    {attribute 'pytmc' := 'pv: TOP:RTD:01'}
    RTD_TOP_1 : FB_CC_TempSensor;
    {attribute 'pytmc' := 'pv: TOP:RTD:02'}
    RTD_TOP_2 : FB_CC_TempSensor;
    {attribute 'pytmc' := 'pv: BOTTOM:RTD:01'}
    RTD_Bottom_1 : FB_CC_TempSensor;
    {attribute 'pytmc' := 'pv: BOTTOM:RTD:02'}
    RTD_Bottom_2 : FB_CC_TempSensor;
    {attribute 'pytmc' := 'pv: NORTH:RTD:01'}
    RTD_North_1 : FB_CC_TempSensor;
    {attribute 'pytmc' := 'pv: NORTH:RTD:02'}
    RTD_North_2 : FB_CC_TempSensor;
    {attribute 'pytmc' := 'pv: SOUTH:RTD:01'}
    RTD_South_1 : FB_CC_TempSensor;
    {attribute 'pytmc' := 'pv: SOUTH:RTD:02'}
    RTD_South_2 : FB_CC_TempSensor;
    (* PMPS reactive-DB key for the device's allowed temperature. *)
    sPmpsState : STRING;
    fbReadPMPSDB : FB_JsonDocToSafeBP;
    astTempDB    : ARRAY[1..1] OF ST_DbStateParams;
    (* fbReadPMPSDB.bExecute needs a rising edge; a real PMPS file read produces one as bBusy falls.
       Taken as REFERENCE TO so a test can drive its own BOOL and simulate the edge
       instead of reaching into MOTION_GVL.fbPmpsFileReader directly.
    *)
    bFileReaderBusy : REFERENCE TO BOOL;
    (* Margin (mm) subtracted from the authorized width/height when snapping
       the request into PMPS compliance. Set via FB_Init, defaults to 0.01. *)
    fApertureMargin : REAL := 0.01;
END_VAR

IF NOT __ISVALIDREF(THIS^.aiMotionStage)
   OR NOT __ISVALIDREF(THIS^.fbFFHWO) OR NOT __ISVALIDREF(bFileReaderBusy) THEN
    RETURN;
END_IF


// Parent body: EPICS edge-trigger consumption only (no REF touch).
SUPER^();


// Inherited dispatch (parity with legacy FB_SLITS_POWER body
// invoking ACT_CalculatePositions / ACT_Motion).
M_CalculatePositions();
M_Motion();

// PMPS reactive temperature DB lookup. bExecute needs a rising edge,
// produced as the caller-injected file-reader busy flag falls. Guard
// the REF (single condition, no short-circuit hazard) so an unbound
// instance stays inert rather than dereferencing a nil ref.
astTempDB[1].sPmpsState := sPmpsState;
fbReadPMPSDB(
    bExecute    := NOT bFileReaderBusy,
    jsonDoc     := PMPS_GVL.BP_jsonDoc,
    sDeviceName := sDeviceName,
    arrStates   := astTempDB,
    io_fbFFHWO  := fbFFHWO
);

// All 8 RTDs share the same fault threshold (resolved from the DB).
RTD_TOP_1(
    fFaultThreshold := astTempDB[1].stReactiveParams.nTempSP,
    sDevName        := sDeviceName,
    io_fbFFHWO      := fbFFHWO
);
RTD_TOP_2(
    fFaultThreshold := astTempDB[1].stReactiveParams.nTempSP,
    sDevName        := sDeviceName,
    io_fbFFHWO      := fbFFHWO
);
RTD_Bottom_1(
    fFaultThreshold := astTempDB[1].stReactiveParams.nTempSP,
    sDevName        := sDeviceName,
    io_fbFFHWO      := fbFFHWO
);
RTD_Bottom_2(
    fFaultThreshold := astTempDB[1].stReactiveParams.nTempSP,
    sDevName        := sDeviceName,
    io_fbFFHWO      := fbFFHWO
);
RTD_North_1(
    fFaultThreshold := astTempDB[1].stReactiveParams.nTempSP,
    sDevName        := sDeviceName,
    io_fbFFHWO      := fbFFHWO
);
RTD_North_2(
    fFaultThreshold := astTempDB[1].stReactiveParams.nTempSP,
    sDevName        := sDeviceName,
    io_fbFFHWO      := fbFFHWO
);
RTD_South_1(
    fFaultThreshold := astTempDB[1].stReactiveParams.nTempSP,
    sDevName        := sDeviceName,
    io_fbFFHWO      := fbFFHWO
);
RTD_South_2(
    fFaultThreshold := astTempDB[1].stReactiveParams.nTempSP,
    sDevName        := sDeviceName,
    io_fbFFHWO      := fbFFHWO
);

fbFlowSwitch();

(* Records sPmpsState and REF-binds the caller-owned file-reader busy flag;
   aiMotionStage (4 blades), fbFFHWO and sDeviceName are bound by base
   FB_SLITS.FB_Init. Blade wiring runs from CallAfterInit. *)
{attribute 'analysis' := '-33'}
METHOD FB_Init : BOOL
VAR_INPUT
    bInitRetains  : BOOL;
    bInCopyCode   : BOOL;
    aiMotionStage : REFERENCE TO ARRAY[1..4] OF I_MotionStage;
    fbFFHWO       : REFERENCE TO FB_HardwareFFOutput;
    sDeviceName   : STRING;
    sPmpsState 	  : STRING;
    bFileReaderBusy : REFERENCE TO BOOL;
    fApertureMargin : REAL;
END_VAR
THIS^.sPmpsState := sPmpsState;
THIS^.bFileReaderBusy REF= bFileReaderBusy;
THIS^.fApertureMargin := fApertureMargin;
END_METHOD

(* Integrator-driven PMPS aperture-safety reconciliation, called each cycle
   with index = this device's slot in astApertures. Mirrors actual geometry
   into AptArrayStatus, faults FFO when actual gap exceeds the authorized
   envelope (or always, out of PMPS mode), and in PMPS mode snaps the request
   into compliance. Caller must ensure index is valid (no short-circuit). *)
METHOD M_UpdatePMPS : BOOL
VAR_INPUT
    index : INT;
END_VAR
// Mirror current actual aperture geometry and any-blade error state.
THIS^.AptArrayStatus.Height := THIS^.rActApertureSizeY;
THIS^.AptArrayStatus.Width  := THIS^.rActApertureSizeX;
THIS^.AptArrayStatus.xOK    :=
        NOT (THIS^.aiMotionStage[E_SlitsBlade.TOP   ].MotionStatus.bError)
    AND NOT (THIS^.aiMotionStage[E_SlitsBlade.BOTTOM].MotionStatus.bError)
    AND NOT (THIS^.aiMotionStage[E_SlitsBlade.NORTH ].MotionStatus.bError)
    AND NOT (THIS^.aiMotionStage[E_SlitsBlade.SOUTH ].MotionStatus.bError);

// Aperture-envelope evaluation.
IF ( THIS^.rActApertureSizeX > (AptArrayReq.Width  - (2 * ABS(THIS^.rActCenterX)))
     AND PMPS_GVL.stCurrentBeamParameters.astApertures[index].Width  > 0 )
OR ( THIS^.rActApertureSizeY > (AptArrayReq.Height - (2 * ABS(THIS^.rActCenterY)))
     AND PMPS_GVL.stCurrentBeamParameters.astApertures[index].Height > 0 ) THEN
    FFO.i_xOK := FALSE;
ELSE
    FFO.i_xOK := TRUE;
END_IF

IF xPMPSMode THEN
    IF THIS^.rActApertureSizeX > AptArrayReq.Width THEN
        rReqApertureSizeX := AptArrayReq.Width - fApertureMargin;
    END_IF
    IF THIS^.rActApertureSizeY > AptArrayReq.Height THEN
        rReqApertureSizeY := AptArrayReq.Height - fApertureMargin;
    END_IF
ELSE
    FFO.i_xOK := FALSE;
END_IF

FFO(
    i_xAutoReset := TRUE,
    io_fbFFHWO   := fbFFHWO
);
END_METHOD

END_FUNCTION_BLOCK

// ---- Devices/SLITS/FB_SLITS.TcPOU
(* Four-blade slit aperture controller (Top/Bottom/North/South), ND framework.
   Each blade uses a per-cycle FB_StatePTPMove single-shot mover (targets
   recomputed from EPICS aperture width/center + encoder offsets), not a named
   state mover. Caller-owned stages, PMPS FFO and device name injected via FB_Init
   REFERENCE TO; CallAfterInit wires blade interfaces. Motion parameters
   (velocity/accel/decel/jerk) belong to the caller-owned stage, set once at
   commissioning and persisted; FB_SLITS does not apply them. *)
{attribute 'analysis' := '-33'}
{attribute 'call_after_init'}
FUNCTION_BLOCK FB_SLITS
VAR_INPUT
    {attribute 'pytmc' := '
    pv: PMPS_OK
    io: i
    field: ZNAM False
    field: ONAM True
    '}
    bMoveOk : BOOL;

    (* Per-blade encoder zero-offsets (EPICS-settable). *)
    {attribute 'pytmc' := '
    pv: Offset_Top
    io: io
    '}
    rEncoderOffsetTop : REAL;

    {attribute 'pytmc' := '
    pv: ZeroOffset_Bottom
    io: io
    '}
    rEncoderOffsetBottom : REAL;

    {attribute 'pytmc' := '
    pv: ZeroOffset_North
    io: io
    '}
    rEncoderOffsetNorth : REAL;

    {attribute 'pytmc' := '
    pv: ZeroOffset_South
    io: io
    '}
    rEncoderOffsetSouth : REAL;
END_VAR
VAR CONSTANT
    (* Position-compare deltas for the blade ST_PositionState. *)
    fSmallDelta : LREAL := 0.01;
     (* Reference blade motion tuning (velocity/accel/decel/jerk). Not applied
       here: motion parameters belong to the caller-owned stage, set once at
       commissioning and persisted. Kept as commissioning reference values. *)
    // fVelocity     : LREAL := 0.2;
    // fAcceleration : LREAL := 0.8;
    // fDeceleration : LREAL := 0.8;
    // fJerk         : LREAL := 0.0;
END_VAR
VAR
    (* Per-blade scratch ST_PositionState. Static fields seeded here;
       fPosition and bMoveOk are refreshed each cycle in the body. *)
    stTop    : ST_PositionState := (sName := 'Top',    bValid := TRUE, bUseRawCounts := FALSE, fDelta := fSmallDelta);
    stBottom : ST_PositionState := (sName := 'Bottom', bValid := TRUE, bUseRawCounts := FALSE, fDelta := fSmallDelta);
    stNorth  : ST_PositionState := (sName := 'North',  bValid := TRUE, bUseRawCounts := FALSE, fDelta := fSmallDelta);
    stSouth  : ST_PositionState := (sName := 'South',  bValid := TRUE, bUseRawCounts := FALSE, fDelta := fSmallDelta);

    (* Per-blade PTP movers. iMotionStage is wired in CallAfterInit;
       FB_StatePTPMove tolerates a nil interface until then. *)
    {attribute 'pytmc' := 'pv: TOP'}
    fbTop    : FB_StatePTPMove(
        stPositionState := stTop,
        iMotionStage:=0
    );
    {attribute 'pytmc' := 'pv: BOTTOM'}
    fbBottom : FB_StatePTPMove(
        stPositionState := stBottom,
        iMotionStage:=0
    );
    {attribute 'pytmc' := 'pv: NORTH'}
    fbNorth  : FB_StatePTPMove(
        stPositionState := stNorth,
        iMotionStage:=0
    );
    {attribute 'pytmc' := 'pv: SOUTH'}
    fbSouth  : FB_StatePTPMove(
        stPositionState := stSouth,
        iMotionStage:=0
    );

    (* Aperture-math intermediate targets. *)
    fPosTopBlade    : LREAL;
    fPosBottomBlade : LREAL;
    fPosNorthBlade  : LREAL;
    fPosSouthBlade  : LREAL;

    (* EPICS request / actual aperture geometry. *)
    {attribute 'pytmc' := '
    pv: XWID_REQ
    io: io
    '}
    rReqApertureSizeX : REAL;
    {attribute 'pytmc' := '
    pv: YWID_REQ
    io: io
    '}
    rReqApertureSizeY : REAL;
    {attribute 'pytmc' := '
    pv: XCEN_REQ
    io: io
    '}
    rReqCenterX : REAL;
    {attribute 'pytmc' := '
    pv: YCEN_REQ
    io: io
    '}
    rReqCenterY : REAL;

    {attribute 'pytmc' := '
    pv: ACTUAL_XWIDTH
    io: io
    '}
    rActApertureSizeX : REAL;
    {attribute 'pytmc' := '
    pv: ACTUAL_YWIDTH
    io: io
    '}
    rActApertureSizeY : REAL;
    {attribute 'pytmc' := '
    pv: ACTUAL_XCENTER
    io: io
    '}
    rActCenterX : REAL;
    {attribute 'pytmc' := '
    pv: ACTUAL_YCENTER
    io: io
    '}
    rActCenterY : REAL;

    (* Edge-trigger request flags. Cleared on the rising edge each
       cycle but no preset move is dispatched (stub: legacy parity). *)
    {attribute 'pytmc' := '
    pv: OPEN
    io: io
    field: ZNAM False
    field: ONAM True
    '}
    bOpen : BOOL;

    {attribute 'pytmc' := '
    pv: CLOSE
    io: io
    field: ZNAM False
    field: ONAM True
    '}
    bClose : BOOL;

    {attribute 'pytmc' := '
    pv: BLOCK
    io: io
    field: ZNAM False
    field: ONAM True
    '}
    bBlock : BOOL;

    rTrig_Block : R_TRIG;
    rTrig_Open  : R_TRIG;
    rTrig_Close : R_TRIG;

    (* Change-detection latches for EPICS request fields. *)
    rOldReqApertureSizeX : REAL;
    rOldReqApertureSizeY : REAL;
    rOldReqCenterX       : REAL;
    rOldReqCenterY       : REAL;

    bExecuteMotionX : BOOL;
    bExecuteMotionY : BOOL;

    fbLogger : FB_LogMessage := (eSubsystem := E_SubSystem.MOTION);

    (* PMPS aperture-safety fault (driven by FB_SLITS_POWER.M_UpdatePMPS). *)
    FFO : FB_FastFault := (
        i_DevName  := sDeviceName,
        i_Desc     := 'Fault occurs when gaps and/or centers are not within safe margins, or PMPS mode is switched OFF',
        i_TypeCode := 16#FAA
    );

    (* PMPS aperture IO (caller-mapped to terminals). *)
    AptArrayStatus AT %Q* : ST_PMPS_Aperture_IO;
    AptArrayReq    AT %I* : ST_PMPS_Aperture_IO;

    (* REF backing fields, populated by FB_Init. *)
    {attribute 'no_copy'}
    aiMotionStage : REFERENCE TO ARRAY[1..4] OF I_MotionStage;
    {attribute 'no_copy'}
    fbFFHWO       : REFERENCE TO FB_HardwareFFOutput;
    sDeviceName   :  STRING;
    nMotor : UINT;
END_VAR

// Legacy parity: the base body consumes only the EPICS Open / Close /
// Block edge-triggers. Blade init + motion dispatch lives on the
// FB_SLITS_POWER subclass body.
HandleRequests();

(* Auto-fired once after FB_Init binds the REFs. The four FB_StatePTPMove
   blade movers were inline-init'd with nil interface refs, so this re-supplies
   each blade's now-valid interface and scratch ST_PositionState, and sets the
   FFO device name. *)
{attribute 'call_after_init'}
METHOD CallAfterInit
fbTop.CallAfterInit(    stPositionState := stTop,    iMotionStage := aiMotionStage[E_SlitsBlade.TOP]);
fbBottom.CallAfterInit( stPositionState := stBottom, iMotionStage := aiMotionStage[E_SlitsBlade.BOTTOM]);
fbNorth.CallAfterInit(  stPositionState := stNorth,  iMotionStage := aiMotionStage[E_SlitsBlade.NORTH]);
fbSouth.CallAfterInit(  stPositionState := stSouth,  iMotionStage := aiMotionStage[E_SlitsBlade.SOUTH]);

FFO.i_DevName := sDeviceName;
END_METHOD

(* REF-binds caller-owned aiMotionStage (4 blades), fbFFHWO and sDeviceName
   at instantiation. Blade interface wiring runs from CallAfterInit once these
   REFs are bound. *)
{attribute 'analysis' := '-33'}
METHOD FB_Init : BOOL
VAR_INPUT
    bInitRetains  : BOOL;
    bInCopyCode   : BOOL;
    aiMotionStage : REFERENCE TO ARRAY[1..4] OF I_MotionStage;
    fbFFHWO       : REFERENCE TO FB_HardwareFFOutput;
    sDeviceName   : STRING;
END_VAR
THIS^.aiMotionStage REF= aiMotionStage;
THIS^.fbFFHWO       REF= fbFFHWO;
THIS^.sDeviceName   := sDeviceName;
END_METHOD

(*
    Consume the EPICS Open / Close / Block rising-edge requests and
    self-clear the flags. No preset move is dispatched (legacy stub).
*)
METHOD HandleRequests
rTrig_Block(CLK := bBlock);
rTrig_Open(CLK := bOpen);
rTrig_Close(CLK := bClose);

IF rTrig_Block.Q THEN
    bBlock := FALSE;
END_IF
IF rTrig_Open.Q THEN
    bOpen := FALSE;
END_IF
IF rTrig_Close.Q THEN
    bClose := FALSE;
END_IF
END_METHOD

(* Legacy ACT_CalculatePositions equivalent. Detects EPICS request changes
   (rejecting aperture sizes beyond the PMPS-authorized envelope), recomputes
   per-blade targets from requested gap + center + encoder offset, and refreshes
   actual aperture geometry feedback from caller-owned motor positions. *)
METHOD M_CalculatePositions
IF rOldReqApertureSizeX <> rReqApertureSizeX THEN
    IF rReqApertureSizeX <= AptArrayReq.Width THEN
        rOldReqApertureSizeX := rReqApertureSizeX;
        bExecuteMotionX      := TRUE;
        fbLogger(sMsg := 'Requested new X gap.', eSevr := TcEventSeverity.Verbose);
    ELSE
        fbLogger(
            sMsg := 'Requested new X gap is larger than PMPS request.',
            eSevr := TcEventSeverity.Verbose
        );
    END_IF
END_IF

IF rOldReqCenterX <> rReqCenterX THEN
    rOldReqCenterX  := rReqCenterX;
    bExecuteMotionX := TRUE;
    fbLogger(sMsg := 'Requested new X center', eSevr := TcEventSeverity.Verbose);
END_IF

IF rOldReqApertureSizeY <> rReqApertureSizeY THEN
    IF rReqApertureSizeY <= AptArrayReq.Height THEN
        rOldReqApertureSizeY := rReqApertureSizeY;
        bExecuteMotionY      := TRUE;
        fbLogger(sMsg := 'Requested new Y gap.', eSevr := TcEventSeverity.Verbose);
    ELSE
        fbLogger(
            sMsg := 'Requested new Y gap is larger than PMPS request.',
            eSevr := TcEventSeverity.Verbose
        );
    END_IF
END_IF

IF rOldReqCenterY <> rReqCenterY THEN
    rOldReqCenterY  := rReqCenterY;
    bExecuteMotionY := TRUE;
    fbLogger(sMsg := 'Requested new Y center.', eSevr := TcEventSeverity.Verbose);
END_IF

// Per-blade target positions from requested gap + center + per-blade
// encoder offset.
fPosTopBlade    :=  (rReqApertureSizeY / 2) + (rReqCenterY + rEncoderOffsetTop);
fPosBottomBlade := -(rReqApertureSizeY / 2) + (rReqCenterY + rEncoderOffsetBottom);
fPosNorthBlade  :=  (rReqApertureSizeX / 2) + (rReqCenterX + rEncoderOffsetNorth);
fPosSouthBlade  := -(rReqApertureSizeX / 2) + (rReqCenterX + rEncoderOffsetSouth);

// Actual aperture geometry feedback from caller-owned motors.
rActApertureSizeX := LREAL_TO_REAL(
    (aiMotionStage[E_SlitsBlade.NORTH].MotionStatus.fActPosition - rEncoderOffsetNorth)
  - (aiMotionStage[E_SlitsBlade.SOUTH].MotionStatus.fActPosition - rEncoderOffsetSouth)
);
rActApertureSizeY := LREAL_TO_REAL(
    (aiMotionStage[E_SlitsBlade.TOP].MotionStatus.fActPosition    - rEncoderOffsetTop)
  - (aiMotionStage[E_SlitsBlade.BOTTOM].MotionStatus.fActPosition - rEncoderOffsetBottom)
);
rActCenterX := LREAL_TO_REAL(
    ((aiMotionStage[E_SlitsBlade.NORTH].MotionStatus.fActPosition - rEncoderOffsetNorth)
   + (aiMotionStage[E_SlitsBlade.SOUTH].MotionStatus.fActPosition - rEncoderOffsetSouth)) / 2
);
rActCenterY := LREAL_TO_REAL(
    ((aiMotionStage[E_SlitsBlade.TOP].MotionStatus.fActPosition    - rEncoderOffsetTop)
   + (aiMotionStage[E_SlitsBlade.BOTTOM].MotionStatus.fActPosition - rEncoderOffsetBottom)) / 2
);
END_METHOD

(* Legacy ACT_Motion equivalent. Refreshes per-blade ST_PositionState
   fPosition/bMoveOk, asserts bExecute on each FB_StatePTPMove on aperture
   change (self-clears on arrival/error, so re-dispatch waits for completion),
   and ticks the four blade movers cyclically. *)
METHOD M_Motion
stTop.fPosition    := fPosTopBlade;
stTop.bMoveOk      := bMoveOk;

stBottom.fPosition := fPosBottomBlade;
stBottom.bMoveOk   := bMoveOk;

stNorth.fPosition  := fPosNorthBlade;
stNorth.bMoveOk    := bMoveOk;

stSouth.fPosition  := fPosSouthBlade;
stSouth.bMoveOk    := bMoveOk;

IF bExecuteMotionY THEN
    fbTop.bExecute    := TRUE;
    fbBottom.bExecute := TRUE;
END_IF
IF bExecuteMotionX THEN
    fbNorth.bExecute := TRUE;
    fbSouth.bExecute := TRUE;
END_IF
bExecuteMotionX := FALSE;
bExecuteMotionY := FALSE;

fbTop(bMoveOk    := bMoveOk);
fbBottom(bMoveOk := bMoveOk);
fbNorth(bMoveOk  := bMoveOk);
fbSouth(bMoveOk  := bMoveOk);
END_METHOD

(* Set the EPICS aperture request in one call: gap (width/height) and center
   on both axes. M_CalculatePositions picks the values up next cycle and, if a
   field changed and the gap is within the PMPS envelope, dispatches the moves. *)
METHOD SetApertureRequest
VAR_INPUT
    ApertureSizeX : REAL;
    ApertureSizeY : REAL;
    CenterX       : REAL;
    CenterY       : REAL;
END_VAR
rReqApertureSizeX := ApertureSizeX;
rReqApertureSizeY := ApertureSizeY;
rReqCenterX       := CenterX;
rReqCenterY       := CenterY;
END_METHOD

METHOD INTERNAL SetAptWidthHeight
VAR_INPUT
    Width : REAL;
    Height : REAL;
END_VAR
THIS^.AptArrayReq.Width := Width;
THIS^.AptArrayReq.Height := Height;
END_METHOD

END_FUNCTION_BLOCK

// ---- Tests/FB_WFSTest.TcPOU
FUNCTION_BLOCK FB_WFSTest EXTENDS FB_TestSuite
VAR
    (* Caller-owned axis, persistent storage, and Y motor.
       In a real PRG the AxisRef would come from MAIN.Mxx. *)
    axRef    : ARRAY[1..2] OF AXIS_REF;
    fbPDS    : LCLS_Tc_DevAbs.FB_PersistentDataStorage;

    // Z motor (focus adjust).
    fbMotorZ : FB_MotionStageNC(AxisRef := axRef[1], iPersistentDataStorage := fbPDS, sName := 'Z');
    (* FB_WFS is single-axis (nActiveMotorCount := 1), so only slot 1
       holds a real motor. aiMotionStage is sized to
       MotionConstants.MAX_STATE_MOTORS to match FB_WFS.FB_Init's
       fixed-size signature; slots 2-4 default-init to a nil interface
       and are never touched. *)
    fbMotorY : FB_MotionStageNC(AxisRef := axRef[2], iPersistentDataStorage := fbPDS, sName := 'Y');
    aiMotionStage : ARRAY[1..MotionConstants.MAX_STATE_MOTORS] OF I_MotionStage := [fbMotorY];

    {attribute 'pytmc' := '
        pv: MMS
        array: 1..1 | 1..6
    '}
    astPositionState : ARRAY[1..MotionConstants.MAX_STATE_MOTORS]
                         OF ARRAY[1..GeneralConstants.MAX_STATES] OF ST_PositionState;

    fbFFHWO    : FB_HardwareFFOutput;
    fbArbiter  : FB_Arbiter(1);
    fbSubSysIO : FB_DummyArbIO;

    sDeviceName    : STRING := 'TST:WFS';
    sTransitionKey : STRING := 'TST:WFS-TRANSITION';

    (* Caller-owned file-reader status, bound to FB_WFS by REFERENCE
       TO. In a real PRG these point at MOTION_GVL.fbPmpsFileReader;
       here they stay FALSE so the DB read proceeds. *)
    bFileReaderBusy  : BOOL;
    bFileReaderError : BOOL;

    fbWFS : FB_WFS(
        aiMotionStage         := aiMotionStage,
        astPositionState      := astPositionState,
        fbFFHWO               := fbFFHWO,
        fbArbiter             := fbArbiter,
        sDeviceName           := sDeviceName,
        sTransitionKey        := sTransitionKey,
        bEnableBeamParams     := TRUE,
        bEnablePositionLimits := TRUE,
        bReadDBNow            := TRUE,
        bFileReaderBusy       := bFileReaderBusy,
        bFileReaderError      := bFileReaderError
    );

    (* Per-install PMPS-side state config (caller-owned). Mirrors what
       a real PRG_xxL0_WFS would declare. stDefault is the caller-owned
       baseline template that FB_CC_StatePMPSConfig's inner FB_StateSetup
       preloads from; fbWFS subsequently overrides per-state sName and
       fDelta via its own FB_CC_InternalStateConfig array. *)
    stDefault : ST_PositionState := (
        bMoveOk       := TRUE,
        bValid        := TRUE,
        bUseRawCounts := FALSE
    );

    afbStatePMPS : ARRAY[1..6] OF FB_CC_StatePMPSConfig[
        (stPositionState := astPositionState[1][E_WFS_States.OUT],
         stDefault       := stDefault,
         fPosition       := 10,
         sPmpsState      := 'TST:WFS-OUT'),
        (stPositionState := astPositionState[1][E_WFS_States.TARGET1],
         stDefault       := stDefault,
         fPosition       := 20,
         sPmpsState      := 'TST:WFS-TARGET1'),
        (stPositionState := astPositionState[1][E_WFS_States.TARGET2],
         stDefault       := stDefault,
         fPosition       := 30,
         sPmpsState      := 'TST:WFS-TARGET2'),
        (stPositionState := astPositionState[1][E_WFS_States.TARGET3],
         stDefault       := stDefault,
         fPosition       := 40,
         sPmpsState      := 'TST:WFS-TARGET3'),
        (stPositionState := astPositionState[1][E_WFS_States.TARGET4],
         stDefault       := stDefault,
         fPosition       := 50,
         sPmpsState      := 'TST:WFS-TARGET4'),
        (stPositionState := astPositionState[1][E_WFS_States.TARGET5],
         stDefault       := stDefault,
         fPosition       := 60,
         sPmpsState      := 'TST:WFS-TARGET5')
    ];

    bFirstScan : BOOL := TRUE;
    i          : UINT;
END_VAR

(* Fake PMPS handling. *)
fbSubSysIO(
    LA  := fbArbiter,
    FFO := fbFFHWO
);

IF bFirstScan THEN
    fbMotorY.SetModeEnableLimits(
        LimBackward    := TRUE,
        LimForward     := TRUE,
        HomeEnable     := FALSE,
        BrakeMode      := E_StageBrakeMode.IF_ENABLED,
        EnableMode     := E_StageEnableMode.DURING_MOTION,
        HomeMode       := E_EpicsHomeCmd.LOW_LIMIT,
        UserEnable     := TRUE,
        HardwareEnable := TRUE
    );
    fbMotorZ.SetModeEnableLimits(
        LimBackward    := TRUE,
        LimForward     := TRUE,
        HomeEnable     := FALSE,
        BrakeMode      := E_StageBrakeMode.IF_ENABLED,
        EnableMode     := E_StageEnableMode.DURING_MOTION,
        HomeMode       := E_EpicsHomeCmd.LOW_LIMIT,
        UserEnable     := TRUE,
        HardwareEnable := TRUE
    );
    fbMotorZ.SetVelocity(Velocity := 15.5);
    fbMotorZ.RestoreMotionParams      := FALSE;
    fbMotorZ.DoNotRestoreNcParameters := TRUE;
    fbMotorY.SetVelocity(Velocity := 15.5);
    fbMotorY.RestoreMotionParams      := FALSE;
    fbMotorY.DoNotRestoreNcParameters := TRUE;
    bFileReaderBusy  := TRUE;
    bFileReaderError := FALSE;
    bFirstScan := FALSE;
END_IF

fbPDS();
fbMotorY();
fbMotorZ();
fbWFS();
fbSubSysIO(LA := fbArbiter, FFO := fbFFHWO);
bFileReaderBusy  := FALSE;
bFileReaderError := FALSE;

TestStateMove();
TestTempFFO();

METHOD SetWFSTemp
VAR_INPUT
    iTempC : INT;
END_VAR
VAR
    ptr : POINTER TO INT;
END_VAR
ptr  := ADR(fbWFS.fbThermoCouple1.iRaw);
ptr^ := iTempC * 10;

ptr  := ADR(fbWFS.fbThermoCouple2.iRaw);
ptr^ := iTempC * 10;
END_METHOD

(*
    Smoke test for WFS state-move wiring. Walks OUT then TARGET1 and
    asserts each lands within fTolerance of the configured fPosition.
    Mirrors FB_REFTest: stageReady gate up front, NOT bMoving +
    position-tolerance check per state, 60s watchdog, on timeout
    AssertTrue(FALSE, ...) with the current step and observed
    position. Two moves is enough to exercise the FB wiring; the
    motion stack itself is covered by the
    lcls-twincat-motion-abstraction test suite.
*)
METHOD TestStateMove
VAR_INST
    tonTimer  : TON;
    nTestStep : INT := 0;
    fObserved : LREAL;
END_VAR
VAR CONSTANT
    fTolerance : LREAL := 2.0;
END_VAR
TEST('TestWFSStateMove');

tonTimer(IN := TRUE, PT := T#60s);
fObserved := fbMotorY.stMotionStatus.fActPosition;

CASE nTestStep OF
    0:
        IF fbMotorY.stMotionStatus.bStageReady
           AND NOT fbMotorY.stMotionStatus.bError THEN
            fbWFS.eEnumSet := E_WFS_States.OUT;
            nTestStep      := 1;
        END_IF
    1:
        (* OUT is configured at fPosition := 10 in afbStatePMPS[1]. *)
        IF fbWFS.eEnumGet = E_WFS_States.OUT
           AND NOT fbMotorY.stMotionStatus.bMoving
           AND ABS(fObserved - 10.0) <= fTolerance THEN
            fbWFS.eEnumSet := E_WFS_States.TARGET1;
            nTestStep      := 2;
        END_IF
    2:
        (* TARGET1 is configured at fPosition := 20 in afbStatePMPS[2]. *)
        IF fbWFS.eEnumGet = E_WFS_States.TARGET1
           AND NOT fbMotorY.stMotionStatus.bMoving
           AND ABS(fObserved - 20.0) <= fTolerance THEN
            AssertTrue(
                Condition := TRUE,
                Message   := 'TestWFSStateMove: OUT then TARGET1 reached within tolerance');
            nTestStep := 3;
        END_IF
END_CASE

IF nTestStep = 3 THEN
    TEST_FINISHED();
ELSIF tonTimer.Q THEN
    AssertTrue(
        Condition := FALSE,
        Message   := CONCAT(
            CONCAT(
                CONCAT('TestWFSStateMove: timed out at step ', TO_STRING(nTestStep)),
                CONCAT(', eEnumGet=', TO_STRING(TO_UDINT(fbWFS.eEnumGet)))),
            CONCAT(', fActPos=', TO_STRING(fObserved))));
    TEST_FINISHED();
END_IF
END_METHOD

METHOD TestTempFFO
VAR_INST
    tonTimer    : TON;
    nStep       : UINT := 0;
    bOutChecked : BOOL := FALSE;
    bInChecked  : BOOL := FALSE;
END_VAR
VAR CONSTANT
    nLastStep : UINT := 3;
END_VAR

(* Do we fault at the correct times?
   Parasitically depends on state move test. *)
TEST('TestWFSTempFFO');

(* Prepare a timeout *)
tonTimer(IN := TRUE, PT := T#10s);

CASE nStep OF
    0:
        (* Set both thermocouple temperatures to crazy high number. *)
        SetWFSTemp(100);
        nStep := nStep + 1;
    1:
        (* Wait till we see "OUT" state and one other state (OUT
           should be no fault). *)
        IF fbWFS.eEnumGet = E_WFS_States.OUT THEN
            AssertTrue(
                fbWFS.fbThermoCouple1.FFO.i_xOK,
                'TC1 faulted even in out position!'
            );
            AssertTrue(
                fbWFS.fbThermoCouple2.FFO.i_xOK,
                'TC2 faulted even in out position!'
            );
            bOutChecked := TRUE;
        ELSIF fbWFS.eEnumGet <> E_WFS_States.Unknown THEN
            AssertFalse(
                fbWFS.fbThermoCouple1.FFO.i_xOK,
                'TC1 no fault even for an in position!'
            );
            AssertFalse(
                fbWFS.fbThermoCouple2.FFO.i_xOK,
                'TC2 no fault even for an in position!'
            );
            bInChecked := TRUE;
        END_IF
        IF bOutChecked AND bInChecked THEN
            nStep := nStep + 1;
        END_IF
    2:
        (* Set both thermocouple temperatures to low again. *)
        SetWFSTemp(0);
        nStep := nStep + 1;
    3:
        AssertTrue(
            fbWFS.fbThermoCouple1.FFO.i_xOK,
            'TC1 faulted even with low temp!'
        );
        AssertTrue(
            fbWFS.fbThermoCouple2.FFO.i_xOK,
            'TC2 faulted even with low temp!'
        );
        nStep := nStep + 1;
END_CASE

IF tonTimer.Q OR nStep > nLastStep THEN
    AssertFalse(tonTimer.Q, 'Timeout in WFS temp FFO test');
    TEST_FINISHED();
END_IF
END_METHOD

END_FUNCTION_BLOCK

// ---- Devices/WFS/FB_WFS.TcPOU
(* WaveFront Sensor target (WFS): thin ND-framework state-mover wrapper.
   Y mover via FB_PositionStatePMPSND (states OUT, TARGET1..TARGET5), plus a
   tick site for two in-beam thermocouples (state-gated), a flow switch (FEE)
   and a flow meter (hutch). Caller-owned deps injected via FB_Init REFERENCE
   TO and forwarded to fbStates; enum bridge and toggles re-forwarded each cycle. *)
{attribute 'call_after_init'}
FUNCTION_BLOCK FB_WFS
VAR_INPUT
    // Set this to a non-unknown value to request a new move.
    {attribute 'pytmc' := '
        pv: MMS:STATE:SET
        io: io
    '}
    eEnumSet : E_WFS_States;
END_VAR
VAR
    {attribute 'pytmc' := 'pv: STC:01'}
    fbThermoCouple1 : FB_CC_TempSensor;

    {attribute 'pytmc' := 'pv: STC:02'}
    fbThermoCouple2 : FB_CC_TempSensor;

    {attribute 'pytmc' := 'pv: FSW'}
    fbFlowSwitch : FB_XTES_Flowswitch;

    {attribute 'pytmc' := 'pv: FWM'}
    fbFlowMeter : FB_AnalogInput := (iTermBits := 15, fTermMax := 60, fTermMin := 0);

    (* REFERENCE TO backing fields populated by FB_Init. *)
    {attribute 'no_copy'}
    aiMotionStage         : REFERENCE TO ARRAY[1..MotionConstants.MAX_STATE_MOTORS] OF I_MotionStage;
    {attribute 'no_copy'}
    astPositionState      : REFERENCE TO ARRAY[1..MotionConstants.MAX_STATE_MOTORS]
                                            OF ARRAY[1..GeneralConstants.MAX_STATES] OF ST_PositionState;
    {attribute 'no_copy'}
    fbFFHWO               : REFERENCE TO FB_HardwareFFOutput;
    {attribute 'no_copy'}
    fbArbiter             : REFERENCE TO FB_Arbiter;
    sDeviceName           : STRING;
    sTransitionKey        : STRING;
    bEnableMotion         : BOOL := TRUE;
    bEnableBeamParams     : BOOL;
    bEnablePositionLimits : BOOL;
    bReadDBNow            : BOOL;

    bFileReaderBusy       : REFERENCE TO BOOL;
    bFileReaderError      : REFERENCE TO BOOL;

    (* One configurator per WFS state (OUT + 5 targets). Writes the
       per-state sName and fDelta. Ticked cyclically in the body AFTER
       fbStates so its writes win over the template baseline
       FB_StateSetup applied via FB_CC_StatePMPSConfig. Idempotent once
       stPositionState.bUpdated trips. *)
    afbStateDefaults : ARRAY[1..6] OF FB_CC_InternalStateConfig[
        (stPositionState := astPositionState[1][E_WFS_States.OUT],
         sName           := 'OUT',
         fDelta          := FDELTA_DEFAULT),
        (stPositionState := astPositionState[1][E_WFS_States.TARGET1],
         sName           := 'TARGET1',
         fDelta          := FDELTA_DEFAULT),
        (stPositionState := astPositionState[1][E_WFS_States.TARGET2],
         sName           := 'TARGET2',
         fDelta          := FDELTA_DEFAULT),
        (stPositionState := astPositionState[1][E_WFS_States.TARGET3],
         sName           := 'TARGET3',
         fDelta          := FDELTA_DEFAULT),
        (stPositionState := astPositionState[1][E_WFS_States.TARGET4],
         sName           := 'TARGET4',
         fDelta          := FDELTA_DEFAULT),
        (stPositionState := astPositionState[1][E_WFS_States.TARGET5],
         sName           := 'TARGET5',
         fDelta          := FDELTA_DEFAULT)
    ];

    {attribute 'pytmc' := '
        pv: MMS
    '}
    fbStates : FB_PositionStatePMPSND(
        aiMotionStage         := aiMotionStage,
        astPositionState      := astPositionState,
        nActiveMotorCount     := 1,
        eEnumSet              := eEnumSet,
        eEnumGet              := eEnumGet,
        bEnableMotion         := bEnableMotion,
        eMotionRequestPolicy  := E_MotionRequestPolicy.INTERRUPT,
        bEnableBeamParams     := bEnableBeamParams,
        bEnablePositionLimits := bEnablePositionLimits,
        bReadDBNow            := bReadDBNow,
        bFileReaderBusy       := bFileReaderBusy,
        bFileReaderError      := bFileReaderError,
        fbFFHWO               := fbFFHWO,
        fbArbiter             := fbArbiter,
        sDeviceName           := sDeviceName,
        sTransitionKey        := sTransitionKey
    );
    i : UINT;
END_VAR
VAR_OUTPUT
    // The current position state as an enum.
    {attribute 'pytmc' := '
        pv: MMS:STATE:GET
        io: i
    '}
    eEnumGet: E_WFS_States;
    // The PMPS database lookup associated with the current position state.
    stDbStateParams: ST_DbStateParams;
END_VAR
VAR CONSTANT
    (* WFS-wide default tolerance for state in-position detection,
       applied per-state by afbStateDefaults. *)
    FDELTA_DEFAULT : LREAL := 2;
END_VAR

IF NOT __ISVALIDREF(aiMotionStage)
   OR NOT __ISVALIDREF(astPositionState)
   OR NOT __ISVALIDREF(fbFFHWO)
   OR NOT __ISVALIDREF(fbArbiter) THEN
    RETURN;
END_IF

(* Device-side per-state defaults (afbStateDefaults) are written
   once in FB_CC_InternalStateConfig.CallAfterInit; no cyclic tick. *)
fbStates(stDbStateParams=> stDbStateParams);

(* In-beam thermocouples: only fault when something is actually in the
   beam (i.e. not OUT). Driven by the PMPS DB temp setpoint. *)
fbThermoCouple1(
    fFaultThreshold := fbStates.stDbStateParams.stReactiveParams.nTempSP,
    bVeto           := eEnumGet = E_WFS_States.OUT,
    sDevName        := sDeviceName,
    io_fbFFHWO      := fbFFHWO
);
fbThermoCouple2(
    fFaultThreshold := fbStates.stDbStateParams.stReactiveParams.nTempSP,
    bVeto           := eEnumGet = E_WFS_States.OUT,
    sDevName        := sDeviceName,
    io_fbFFHWO      := fbFFHWO
);

fbFlowSwitch();
fbFlowMeter();

(* Auto-fired after FB_Init. fbStates' inline-init ran first and
   forwarded nil refs, so this re-supplies the now-valid refs via
   fbStates.CallAfterInitStateMover / CallAfterInitPMPS and writes the
   per-state device defaults. *)
{attribute 'call_after_init'}
METHOD CallAfterInit
afbStateDefaults[1].CallAfterInit(stPositionState := THIS^.astPositionState[1][E_WFS_States.OUT]);
afbStateDefaults[2].CallAfterInit(stPositionState := THIS^.astPositionState[1][E_WFS_States.TARGET1]);
afbStateDefaults[3].CallAfterInit(stPositionState := THIS^.astPositionState[1][E_WFS_States.TARGET2]);
afbStateDefaults[4].CallAfterInit(stPositionState := THIS^.astPositionState[1][E_WFS_States.TARGET3]);
afbStateDefaults[5].CallAfterInit(stPositionState := THIS^.astPositionState[1][E_WFS_States.TARGET4]);
afbStateDefaults[6].CallAfterInit(stPositionState := THIS^.astPositionState[1][E_WFS_States.TARGET5]);

THIS^.fbStates.CallAfterInitStateMover(
    aiMotionStage         := aiMotionStage,
    astPositionState      := astPositionState,
    nActiveMotorCount     := 1,
    eEnumSet              := eEnumSet,
    eEnumGet              := eEnumGet,
    bEnableMotion         := bEnableMotion,
    eMotionRequestPolicy  := E_MotionRequestPolicy.INTERRUPT,
);

THIS^.fbStates.CallAfterInitPMPS(
    aiMotionStage         := aiMotionStage,
    astPositionState      := astPositionState,
    bEnableBeamParams     := bEnableBeamParams,
    bEnablePositionLimits := bEnablePositionLimits,
    bReadDBNow            := bReadDBNow,
    bFileReaderBusy       := bFileReaderBusy,
    bFileReaderError      := bFileReaderError,
    fbFFHWO               := fbFFHWO,
    fbArbiter             := fbArbiter,
    sDeviceName           := sDeviceName,
    sTransitionKey        := sTransitionKey
);
END_METHOD

(* Stores FB_Init inputs into instance fields; every non-value input is
   REFERENCE TO, REF= bound for the FB lifetime. fbStates inline-init
   captured these params at construction, so this records the same refs
   on THIS^ for body use and live caller writes. *)
{attribute 'analysis' := '-33'}
METHOD FB_Init : BOOL
VAR_INPUT
    bInitRetains     : BOOL;
    bInCopyCode      : BOOL;
    aiMotionStage    : REFERENCE TO ARRAY[1..MotionConstants.MAX_STATE_MOTORS] OF I_MotionStage;
    astPositionState : REFERENCE TO ARRAY[1..MotionConstants.MAX_STATE_MOTORS]
                                       OF ARRAY[1..GeneralConstants.MAX_STATES] OF ST_PositionState;
    fbFFHWO          : REFERENCE TO FB_HardwareFFOutput;
    fbArbiter        : REFERENCE TO FB_Arbiter;
    sDeviceName      : STRING;
    sTransitionKey   : STRING;
    bEnableBeamParams      : BOOL;
    bEnablePositionLimits  : BOOL;
    bReadDBNow             : BOOL;
    bFileReaderBusy       : REFERENCE TO BOOL;
    bFileReaderError      : REFERENCE TO BOOL;
END_VAR
THIS^.aiMotionStage    REF= aiMotionStage;
THIS^.astPositionState REF= astPositionState;
THIS^.fbFFHWO          REF= fbFFHWO;
THIS^.fbArbiter        REF= fbArbiter;
THIS^.sDeviceName      := sDeviceName;
THIS^.sTransitionKey   := sTransitionKey;
THIS^.bEnableBeamParams     := bEnableBeamParams;
THIS^.bEnablePositionLimits := bEnablePositionLimits;
THIS^.bReadDBNow            := bReadDBNow;
THIS^.bFileReaderBusy       REF= bFileReaderBusy;
THIS^.bFileReaderError      REF= bFileReaderError;
END_METHOD

END_FUNCTION_BLOCK

// ---- Tests/FB_XPIMTest.TcPOU
FUNCTION_BLOCK FB_XPIMTest EXTENDS FB_TestSuite
VAR
    (* Caller-owned axis, persistent storage, and Y motor.
       In a real PRG the AxisRef would come from MAIN.Mxx. *)
    axRef    : ARRAY[1..3] OF AXIS_REF;
    fbPDS    : LCLS_Tc_DevAbs.FB_PersistentDataStorage;

    fbZoom: FB_MotionStageNC(AxisRef := axRef[1], iPersistentDataStorage := fbPDS, sName := 'Zoom');;
    fbFocus: FB_MotionStageNC(AxisRef := axRef[2], iPersistentDataStorage := fbPDS, sName := 'Focus');;

    (* FB_XPIM is single-axis (nActiveMotorCount := 1), so only slot 1
       holds a real motor. aiMotionStage is sized to
       MotionConstants.MAX_STATE_MOTORS to match FB_XPIM.FB_Init's
       fixed-size signature; slots 2-4 default-init to a nil interface
       and are never touched. *)
    fbMotorY : FB_MotionStageNC(AxisRef := axRef[3], iPersistentDataStorage := fbPDS, sName := 'Y');
    aiMotionStage : ARRAY[1..MotionConstants.MAX_STATE_MOTORS] OF I_MotionStage := [fbMotorY];

    {attribute 'pytmc' := '
        pv: MMS
        astPositionState.array: 1..4
    '}
    astPositionState : ARRAY[1..MotionConstants.MAX_STATE_MOTORS]
                         OF ARRAY[1..GeneralConstants.MAX_STATES] OF ST_PositionState;

    fbFFHWO    : FB_HardwareFFOutput;
    fbArbiter  : FB_Arbiter(1);
    fbSubSysIO : FB_DummyArbIO;

    (* EL6 serial terminal buffers, caller-owned. In a real PRG these
       would be linked to physical EL6xxx terminal IO; here they are
       just standalone locals so the FB_XPIM.FB_Init REFERENCE TO
       inputs have something to bind. *)
    stEl6In  : EL6inData22b;
    stEl6Out : EL6outData22b;

    sDeviceName    : STRING := 'TST:XPIM';
    sTransitionKey : STRING := 'TST:XPIM-TRANSITION';

    (* Caller-owned file-reader status, bound to FB_XPIM by REFERENCE
       TO. In a real PRG these point at MOTION_GVL.fbPmpsFileReader;
       here they stay FALSE so the DB read proceeds. *)
    bFileReaderBusy  : BOOL;
    bFileReaderError : BOOL;

    fbXPIM : FB_XPIM(
        aiMotionStage         := aiMotionStage,
        astPositionState      := astPositionState,
        fbFFHWO               := fbFFHWO,
        fbArbiter             := fbArbiter,
        sDeviceName           := sDeviceName,
        sTransitionKey        := sTransitionKey,
        bEnableBeamParams     := TRUE,
        bEnablePositionLimits := TRUE,
        bReadDBNow            := TRUE,
        bFileReaderBusy       := bFileReaderBusy,
        bFileReaderError      := bFileReaderError,
        stEl6In               := stEl6In,
        stEl6Out              := stEl6Out
    );

    (* Per-install PMPS-side state config (caller-owned). Mirrors what
       a real PRG_xxL0_XPIM would declare. stDefault is the caller-owned
       baseline template that FB_CC_StatePMPSConfig's inner FB_StateSetup
       preloads from; fbXPIM subsequently overrides per-state sName and
       fDelta via its own FB_CC_InternalStateConfig array. *)
    stDefault : ST_PositionState := (
        bMoveOk       := TRUE,
        bValid        := TRUE,
        bUseRawCounts := FALSE
    );

    afbStatePMPS : ARRAY[1..4] OF FB_CC_StatePMPSConfig[
        (stPositionState := astPositionState[1][E_XPIM_States.OUT],
         stDefault       := stDefault,
         fPosition       := 10,
         sPmpsState      := 'TST:XPIM-OUT'),
        (stPositionState := astPositionState[1][E_XPIM_States.YAG],
         stDefault       := stDefault,
         fPosition       := 20,
         sPmpsState      := 'TST:XPIM-YAG'),
        (stPositionState := astPositionState[1][E_XPIM_States.DIAMOND],
         stDefault       := stDefault,
         fPosition       := 30,
         sPmpsState      := 'TST:XPIM-DIAMOND'),
        (stPositionState := astPositionState[1][E_XPIM_States.RETICLE],
         stDefault       := stDefault,
         fPosition       := 40,
         sPmpsState      := 'TST:XPIM-RETICLE')
    ];

    bFirstScan : BOOL := TRUE;
    i          : UINT;
END_VAR

(* Fake PMPS handling. *)
fbSubSysIO(
    LA  := fbArbiter,
    FFO := fbFFHWO
);

IF bFirstScan THEN
    fbMotorY.SetModeEnableLimits(
        LimBackward    := TRUE,
        LimForward     := TRUE,
        HomeEnable     := FALSE,
        BrakeMode      := E_StageBrakeMode.IF_ENABLED,
        EnableMode     := E_StageEnableMode.DURING_MOTION,
        HomeMode       := E_EpicsHomeCmd.LOW_LIMIT,
        UserEnable     := TRUE,
        HardwareEnable := TRUE
    );
    fbZoom.SetModeEnableLimits(
        LimBackward    := TRUE,
        LimForward     := TRUE,
        HomeEnable     := FALSE,
        BrakeMode      := E_StageBrakeMode.IF_ENABLED,
        EnableMode     := E_StageEnableMode.DURING_MOTION,
        HomeMode       := E_EpicsHomeCmd.LOW_LIMIT,
        UserEnable     := TRUE,
        HardwareEnable := TRUE
    );
    fbFocus.SetModeEnableLimits(
        LimBackward    := TRUE,
        LimForward     := TRUE,
        HomeEnable     := FALSE,
        BrakeMode      := E_StageBrakeMode.IF_ENABLED,
        EnableMode     := E_StageEnableMode.DURING_MOTION,
        HomeMode       := E_EpicsHomeCmd.LOW_LIMIT,
        UserEnable     := TRUE,
        HardwareEnable := TRUE
    );
    fbMotorY.SetVelocity(Velocity := 15.5);
    fbMotorY.RestoreMotionParams      := FALSE;
    fbMotorY.DoNotRestoreNcParameters := TRUE;
    fbZoom.SetVelocity(Velocity := 15.5);
    fbZoom.RestoreMotionParams      := FALSE;
    fbZoom.DoNotRestoreNcParameters := TRUE;
    fbFocus.SetVelocity(Velocity := 15.5);
    fbFocus.RestoreMotionParams      := FALSE;
    fbFocus.DoNotRestoreNcParameters := TRUE;
    bFileReaderBusy  := TRUE;
    bFileReaderError := FALSE;
    bFirstScan := FALSE;
END_IF

fbPDS();
fbMotorY();
fbZoom();
fbFocus();
fbXPIM();

TestStateMove();

bFileReaderBusy  := FALSE;
bFileReaderError := FALSE;

(*
    Smoke test for XPIM state-move wiring. Walks OUT then YAG and
    asserts each lands within fTolerance of the configured fPosition.
    Mirrors FB_REFTest: stageReady gate up front, NOT bMoving +
    position-tolerance check per state, 60s watchdog, on timeout
    AssertTrue(FALSE, ...) with the current step and observed
    position. Two moves is enough to exercise the FB wiring; the
    motion stack itself is covered by the
    lcls-twincat-motion-abstraction test suite.
*)
METHOD TestStateMove
VAR_INST
    tonTimer  : TON;
    nTestStep : INT := 0;
    fObserved : LREAL;
END_VAR
VAR CONSTANT
    fTolerance : LREAL := 2.0;
END_VAR
TEST('TestXPIMStateMove');

tonTimer(IN := TRUE, PT := T#60s);
fObserved := fbMotorY.stMotionStatus.fActPosition;

CASE nTestStep OF
    0:
        IF fbMotorY.stMotionStatus.bStageReady
           AND NOT fbMotorY.stMotionStatus.bError THEN
            fbXPIM.eEnumSet := E_XPIM_States.OUT;
            nTestStep       := 1;
        END_IF
    1:
        (* OUT is configured at fPosition := 10 in afbStatePMPS[1]. *)
        IF fbXPIM.eEnumGet = E_XPIM_States.OUT
           AND NOT fbMotorY.stMotionStatus.bMoving
           AND ABS(fObserved - 10.0) <= fTolerance THEN
            fbXPIM.eEnumSet := E_XPIM_States.YAG;
            nTestStep       := 2;
        END_IF
    2:
        (* YAG is configured at fPosition := 20 in afbStatePMPS[2]. *)
        IF fbXPIM.eEnumGet = E_XPIM_States.YAG
           AND NOT fbMotorY.stMotionStatus.bMoving
           AND ABS(fObserved - 20.0) <= fTolerance THEN
            AssertTrue(
                Condition := TRUE,
                Message   := 'TestXPIMStateMove: OUT then YAG reached within tolerance');
            nTestStep := 3;
        END_IF
END_CASE

IF nTestStep = 3 THEN
    TEST_FINISHED();
ELSIF tonTimer.Q THEN
    AssertTrue(
        Condition := FALSE,
        Message   := CONCAT(
            CONCAT(
                CONCAT('TestXPIMStateMove: timed out at step ', TO_STRING(nTestStep)),
                CONCAT(', eEnumGet=', TO_STRING(TO_UDINT(fbXPIM.eEnumGet)))),
            CONCAT(', fActPos=', TO_STRING(fObserved))));
    TEST_FINISHED();
END_IF
END_METHOD

END_FUNCTION_BLOCK

// ---- Devices/XPIM/FB_XPIM.TcPOU
(* XTES Profile Imager (XPIM): thin ND-framework state-mover wrapper.
   Y mover via FB_PositionStatePMPSND (states OUT, YAG, DIAMOND, RETICLE),
   plus a tick site for the serial filter wheel, Opal camera power, LED
   (state-gated) and flow switch. Caller-owned deps, incl. EL6 serial buffers,
   injected via FB_Init REFERENCE TO and forwarded to fbStates each cycle. *)
{attribute 'call_after_init'}
FUNCTION_BLOCK FB_XPIM
VAR_INPUT
    // Set this to a non-unknown value to request a new move.
    {attribute 'pytmc' := '
        pv: MMS:STATE:SET
        io: io
    '}
    eEnumSet : E_XPIM_States;
END_VAR
VAR

    {attribute 'pytmc' := 'pv: MFW'}
    fbFilterWheel : FB_XPIM_FilterWheel;

    {attribute 'pytmc' := 'pv: CAM'}
    fbOpal : FB_XPIM_Opal;

    {attribute 'pytmc' := 'pv: CIL'}
    fbLED : FB_XPIM_LED;

    {attribute 'pytmc' := 'pv: FSW'}
    fbFlowSwitch : FB_XTES_Flowswitch;

    (* REFERENCE TO backing fields populated by FB_Init.*)
    {attribute 'no_copy'}
    aiMotionStage         : REFERENCE TO ARRAY[1..MotionConstants.MAX_STATE_MOTORS] OF I_MotionStage;
    {attribute 'no_copy'}
    astPositionState      : REFERENCE TO ARRAY[1..MotionConstants.MAX_STATE_MOTORS]
                                            OF ARRAY[1..GeneralConstants.MAX_STATES] OF ST_PositionState;
    {attribute 'no_copy'}
    fbFFHWO               : REFERENCE TO FB_HardwareFFOutput;
    {attribute 'no_copy'}
    fbArbiter             : REFERENCE TO FB_Arbiter;
    sDeviceName           : STRING;
    sTransitionKey        : STRING;
    bEnableMotion         : BOOL := TRUE;
    bEnableBeamParams     : BOOL;
    bEnablePositionLimits : BOOL;
    bReadDBNow            : BOOL;
    {attribute 'no_copy'}
    bFileReaderBusy       : REFERENCE TO BOOL;
    {attribute 'no_copy'}
    bFileReaderError      : REFERENCE TO BOOL;

    fbStates : FB_PositionStatePMPSND(
        aiMotionStage         := aiMotionStage,
        astPositionState      := astPositionState,
        nActiveMotorCount     := 1,
        eEnumSet              := eEnumSet,
        eEnumGet              := eEnumGet,
        bEnableMotion         := bEnableMotion,
        eMotionRequestPolicy  := E_MotionRequestPolicy.INTERRUPT,
        bEnableBeamParams     := bEnableBeamParams,
        bEnablePositionLimits := bEnablePositionLimits,
        bReadDBNow            := bReadDBNow,
        bFileReaderBusy       := bFileReaderBusy,
        bFileReaderError      := bFileReaderError,
        fbFFHWO               := fbFFHWO,
        fbArbiter             := fbArbiter,
        sDeviceName           := sDeviceName,
        sTransitionKey        := sTransitionKey
    );

    (* EL6 serial terminal buffers, caller-owned and physically linked
       to the EL6xxx terminal IO. Passed through to FB_XPIM_FilterWheel
       via VAR_IN_OUT each cycle. *)
    {attribute 'no_copy'}
    stEl6In               : REFERENCE TO EL6inData22b;
    {attribute 'no_copy'}
    stEl6Out              : REFERENCE TO EL6outData22b;

    (* One configurator per XPIM state. Writes the per-state sName and
       fDelta. Ticked cyclically in the body AFTER fbStates so its
       writes win over the template baseline FB_StateSetup applied via
       FB_CC_StatePMPSConfig. Idempotent once
       stPositionState.bUpdated trips. *)
    afbStateDefaults : ARRAY[1..4] OF FB_CC_InternalStateConfig[
        (stPositionState := astPositionState[1][E_XPIM_States.OUT],
         sName           := 'OUT',
         fDelta          := FDELTA_DEFAULT),
        (stPositionState := astPositionState[1][E_XPIM_States.YAG],
         sName           := 'YAG',
         fDelta          := FDELTA_DEFAULT),
        (stPositionState := astPositionState[1][E_XPIM_States.DIAMOND],
         sName           := 'DIAMOND',
         fDelta          := FDELTA_DEFAULT),
        (stPositionState := astPositionState[1][E_XPIM_States.RETICLE],
         sName           := 'RETICLE',
         fDelta          := FDELTA_DEFAULT)
    ];

    i : UINT;
END_VAR
VAR_OUTPUT
    // The current position state as an enum.
    {attribute 'pytmc' := '
        pv: MMS:STATE:GET
        io: i
    '}
    eEnumGet: E_XPIM_States;
    // The PMPS database lookup associated with the current position state.
    stDbStateParams: ST_DbStateParams;
END_VAR

VAR CONSTANT
    (* XPIM-wide default tolerance for state in-position detection,
       applied per-state by afbStateDefaults. *)
    FDELTA_DEFAULT : LREAL := 2;
END_VAR

IF NOT __ISVALIDREF(aiMotionStage)
   OR NOT __ISVALIDREF(astPositionState)
   OR NOT __ISVALIDREF(fbFFHWO)
   OR NOT __ISVALIDREF(fbArbiter)
   OR NOT __ISVALIDREF(stEl6In)
   OR NOT __ISVALIDREF(stEl6Out) THEN
    RETURN;
END_IF

(* Device-side per-state defaults (afbStateDefaults) are written
   once in FB_CC_InternalStateConfig.CallAfterInit; no cyclic tick. *)
fbStates(stDbStateParams=> stDbStateParams);

(* Serial filter wheel: bExecute := TRUE keeps the comm state machine
   running continuously. *)
fbFilterWheel(
    bExecute  := TRUE,
    stIn_EL6  := stEl6In,
    stOut_EL6 := stEl6Out
);

fbOpal();
fbLED(enumXPIM := eEnumGet);
fbFlowSwitch();

(* Auto-fired after FB_Init. fbStates' inline-init ran first and
   forwarded nil refs, so this re-supplies the now-valid refs via
   fbStates.CallAfterInitStateMover / CallAfterInitPMPS and writes the
   per-state device defaults. *)
{attribute 'call_after_init'}
METHOD CallAfterInit
afbStateDefaults[1].CallAfterInit(stPositionState := THIS^.astPositionState[1][E_XPIM_States.OUT]);
afbStateDefaults[2].CallAfterInit(stPositionState := THIS^.astPositionState[1][E_XPIM_States.YAG]);
afbStateDefaults[3].CallAfterInit(stPositionState := THIS^.astPositionState[1][E_XPIM_States.DIAMOND]);
afbStateDefaults[4].CallAfterInit(stPositionState := THIS^.astPositionState[1][E_XPIM_States.RETICLE]);

THIS^.fbStates.CallAfterInitStateMover(
    aiMotionStage         := aiMotionStage,
    astPositionState      := astPositionState,
    nActiveMotorCount     := 1,
    eEnumSet              := eEnumSet,
    eEnumGet              := eEnumGet,
    bEnableMotion         := bEnableMotion,
    eMotionRequestPolicy  := E_MotionRequestPolicy.INTERRUPT,
);

THIS^.fbStates.CallAfterInitPMPS(
    aiMotionStage         := aiMotionStage,
    astPositionState      := astPositionState,
    bEnableBeamParams     := bEnableBeamParams,
    bEnablePositionLimits := bEnablePositionLimits,
    bReadDBNow            := bReadDBNow,
    bFileReaderBusy       := bFileReaderBusy,
    bFileReaderError      := bFileReaderError,
    fbFFHWO               := fbFFHWO,
    fbArbiter             := fbArbiter,
    sDeviceName           := sDeviceName,
    sTransitionKey        := sTransitionKey
);
END_METHOD

(* Stores FB_Init inputs into instance fields; every non-value input is
   REFERENCE TO, REF= bound for the FB lifetime. fbStates inline-init
   captured these params at construction, so this records the same refs
   on THIS^ for body use and live caller writes. *)
{attribute 'analysis' := '-33'}
METHOD FB_Init : BOOL
VAR_INPUT
    bInitRetains           : BOOL;
    bInCopyCode            : BOOL;
    aiMotionStage          : REFERENCE TO ARRAY[1..MotionConstants.MAX_STATE_MOTORS] OF I_MotionStage;
    astPositionState       : REFERENCE TO ARRAY[1..MotionConstants.MAX_STATE_MOTORS]
                                            OF ARRAY[1..GeneralConstants.MAX_STATES] OF ST_PositionState;
    fbFFHWO                : REFERENCE TO FB_HardwareFFOutput;
    fbArbiter              : REFERENCE TO FB_Arbiter;
    sDeviceName            : STRING;
    sTransitionKey         : STRING;
    bEnableBeamParams      : BOOL;
    bEnablePositionLimits  : BOOL;
    bReadDBNow             : BOOL;
    bFileReaderBusy        : REFERENCE TO BOOL;
    bFileReaderError       : REFERENCE TO BOOL;
    stEl6In                : REFERENCE TO EL6inData22b;
    stEl6Out               : REFERENCE TO EL6outData22b;

END_VAR
THIS^.aiMotionStage    REF= aiMotionStage;
THIS^.astPositionState REF= astPositionState;
THIS^.fbFFHWO          REF= fbFFHWO;
THIS^.fbArbiter        REF= fbArbiter;
THIS^.sDeviceName      := sDeviceName;
THIS^.sTransitionKey   := sTransitionKey;
THIS^.bEnableBeamParams     := bEnableBeamParams;
THIS^.bEnablePositionLimits := bEnablePositionLimits;
THIS^.bReadDBNow            := bReadDBNow;
THIS^.bFileReaderBusy       REF= bFileReaderBusy;
THIS^.bFileReaderError      REF= bFileReaderError;
THIS^.stEl6In          REF= stEl6In;
THIS^.stEl6Out         REF= stEl6Out;
END_METHOD

END_FUNCTION_BLOCK

// ---- Devices/XPIM/FB_XPIM_FilterWheel.TcPOU
FUNCTION_BLOCK FB_XPIM_FilterWheel
VAR_INPUT
    bExecute: BOOL;

    {attribute 'pytmc' := '
        pv: ERR:RESET
        io: output
    '}
    bResetError: BOOL;

    {attribute 'pytmc' := '
        pv: SET
        io: io
    '}
    nSetPos: E_XPIM_Filters;
END_VAR
VAR_OUTPUT
    {attribute 'pytmc' := '
        pv: GET
        io: i
    '}
    nGetPos: E_XPIM_Filters;
    bBusy: BOOL;
    bError: BOOL;
    sError: STRING;
    {attribute 'pytmc' := '
        pv: ERR:MSG
        io: input
    '}
    sLastError: STRING;
    sErrorTS: STRING;
END_VAR
VAR_IN_OUT
    stIn_EL6: EL6inData22B;
    stOut_EL6: EL6outData22B;
END_VAR
VAR
    {attribute 'pytmc' := '
        pv: RAW
    '}
    fbCom: FB_EL6_COM;

    nStep: USINT;
    bIsTest: BOOL;
    fbGetTime: NT_GetTime;
    bStopOnErr: BOOL;
END_VAR

fbCom.sSendSuffix := '$R';
fbCom.sRecvSuffix := '$R';

IF bExecute AND nStep = 0 THEN
    IF bResetError OR NOT bError THEN
        nStep := 10;
    END_IF
ELSIF NOT bExecute THEN
    nStep := 0;
END_IF
CASE nStep OF
    0:
        ; // idle
    10:
        // Get position
        bIsTest := FALSE;
        fbCom(sCmd:='pos?',
            bSend:=TRUE,
            stIn_EL6:=stIn_EL6,
            stOut_EL6:=stOut_EL6);
        nStep := nStep + 10;
    20:
        // Wait for response and set variables
        fbCom(stIn_EL6:=stIn_EL6,
            stOut_EL6:=stOut_EL6);
        IF fbCom.bDone THEN
            bError := FALSE;
            sError := '';
            nGetPos := STRING_TO_USINT(fbCom.sResponse);
            nSetPos := nGetPos;
            nStep := nStep + 10;
            IF nGetPos = 0 THEN
                sError := 'Filter wheel in invalid state';
                bStopOnErr := TRUE;
                nStep := 50;
            END_IF
        END_IF
    30:
        // Wait for a move request
        IF nSetPos <> nGetPos THEN
            fbCom(sCmd:=CONCAT('pos=', UINT_TO_STRING(nSetPos)),
                bSend:=TRUE,
                stIn_EL6:=stIn_EL6,
                stOut_EL6:=stOut_EL6);
            nStep := nStep + 10;
            bBusy := TRUE;
        END_IF
    40:
        fbCom(stIn_EL6:=stIn_EL6,
            stOut_EL6:=stOut_EL6);
        // Wait for move to be done
        IF fbCom.bDone THEN
            bBusy := FALSE;
            nStep := 10;
            // Handle setpoint error
            IF fbCom.sResponse = 'Command error CMD_ARG_INVALID$N$R' THEN
                sError := 'Invalid set position';
                nStep := 50;
            END_IF
        END_IF
    50:
        // Set sError and then jump here for standard handling
        sLastError := sError;
        bError := TRUE;
        fbGetTime(NETID:='',
            START:=TRUE);
        nStep := nStep + 10;
    60:
        // Error handling continued
        fbGetTime();
        IF NOT fbGetTime.BUSY THEN
            sErrorTS := SYSTEMTIME_TO_STRING(fbGetTime.TIMESTR);
            fbGetTime.START := FALSE;
            // set bStopOnErr to TRUE if it was a major error
            IF bStopOnErr THEN
                nStep := 0;
            ELSE
                nStep := 10;
            END_IF
            bStopOnErr := FALSE;
        END_IF
END_CASE
// Check for inner comms errors, report to EPICS same way
IF NOT bError AND
    (fbCom.eRecvErrorID <> COMERROR_NOERROR
    OR fbCom.eSendErrorID <> COMERROR_NOERROR
    OR fbCom.eRecvErrorID <> COMERROR_NOERROR) THEN
    sError := 'Serial Communication Error';
    bStopOnErr := TRUE;
    nStep := 50;
END_IF

END_FUNCTION_BLOCK

// ---- Devices/XPIM/FB_XPIM_Opal.TcPOU
FUNCTION_BLOCK FB_XPIM_Opal
VAR_INPUT
    {attribute 'pytmc' := '
        pv: PWR
        io: io
        field: ZNAM OFF
        field: ONAM ON
    '}
    bOpalPower AT %Q*: BOOL;
END_VAR
VAR
    bOpalInit: BOOL := FALSE;
END_VAR

// Turn the Opal on by default
IF NOT bOpalInit THEN
    bOpalPower := TRUE;
    bOpalInit := TRUE;
END_IF

END_FUNCTION_BLOCK

// ---- Devices/XPIM/FB_XPIM_LED.TcPOU
FUNCTION_BLOCK FB_XPIM_LED
VAR_INPUT
    {attribute 'pytmc' := '
        pv: PWR
        io: io
        field: ZNAM OFF
        field: ONAM ON
    '}
    bLEDPower AT %Q*: BOOL;

    {attribute 'pytmc' := '
        pv: AUTO
        io: io
    '}
    bLEDAuto: BOOL := TRUE;

    {attribute 'pytmc' := '
        pv: CLK:TIMEOUT
        io: io
        field: EGU min
    '}
    fLEDTimeOut: LREAL := 10;

    enumXPIM: E_XPIM_States;
END_VAR
VAR_OUTPUT
    {attribute 'pytmc' := '
        pv: CLK:REMAINING
        io: io
        field: EGU min
    '}
    fLEDRemaining: LREAL;
END_VAR
VAR
    tonLED: TON;
    enumLastCycle: E_XPIM_States := E_XPIM_States.Unknown;
END_VAR

// If configured, change the LED level automatically
// LED is always (and only) useful at Reticle state
IF bLEDAuto AND enumXPIM <> enumLastCycle THEN
    // Turn on the LED when we get to the Reticle
    IF enumXPIM = E_XPIM_States.Reticle THEN
        bLEDPower := TRUE;
    // Turn off the LED when we stop at any other state
    ELSIF enumXPIM <> E_XPIM_States.Unknown THEN
        bLEDPower := FALSE;
    END_IF
END_IF
enumLastCycle := enumXPIM;

// If configured, start a shutdown timer when LED goes high
IF fLEDTimeOut <> 0 THEN;
    tonLED(IN:=bLEDPower,
           PT:=LREAL_TO_TIME(fLEDTimeOut * 60 * 1000));
    fLEDRemaining := fLEDTimeOut - TIME_TO_LREAL(tonLED.ET) / 60 / 1000;

    IF tonLED.Q THEN
        bLEDPower := FALSE;
    END_IF
END_IF

END_FUNCTION_BLOCK

// ---- Tests/FB_CC_TempSensorTest.TcPOU
FUNCTION_BLOCK FB_CC_TempSensorTest EXTENDS FB_TestSuite
VAR
    fbTempSensor: FB_CC_TempSensor;
    fbFFHWO: FB_HardwareFFOutput;
END_VAR


TestBasic();
TestAutoReset();

METHOD SetTempAndRunFB
VAR_INPUT
    iRawTemp: INT;
END_VAR
VAR
    ptr: POINTER TO INT;
END_VAR

ptr := ADR(fbTempSensor.iRaw);
ptr^ := iRawTemp * 10;

fbTempSensor(io_fbFFHWO:=fbFFHWO);
fbFFHWO.ExecuteNoLog();
END_METHOD

METHOD TestAutoReset
VAR_INPUT
END_VAR

TEST('TestAutoReset');

// Set a fixed threshold for the test
fbTempSensor.fFaultThreshold := 30;

// Clear faults
fbTempSensor.bVeto := TRUE;
SetTempAndRunFB(0);
AssertTrue(
    fbFFHWO.astFF[fbTempSensor.FFO.RegistrationIdx].BeamPermitted,
    'Beam not permitted after full clear with low temp',
);

// Cause a fault
fbTempSensor.bVeto := FALSE;
SetTempAndRunFB(100);
AssertFalse(
    fbFFHWO.astFF[fbTempSensor.FFO.RegistrationIdx].BeamPermitted,
    'Beam permitted after high temp',
);

// Remove the fault condition, should still be fauling
fbTempSensor.bVeto := FALSE;
SetTempAndRunFB(0);
AssertFalse(
    fbFFHWO.astFF[fbTempSensor.FFO.RegistrationIdx].BeamPermitted,
    'Beam permitted before manual reset',
);

// Set veto, should no longer be faulting
fbTempSensor.bVeto := TRUE;
SetTempAndRunFB(0);
AssertTrue(
    fbFFHWO.astFF[fbTempSensor.FFO.RegistrationIdx].BeamPermitted,
    'Beam not permitted after veto',
);

TEST_FINISHED();
END_METHOD

METHOD TestBasic

TEST('TestBasic');

fbTempSensor.fFaultThreshold := 10;
fbTempSensor.bVeto := FALSE;
SetTempAndRunFB(2);
AssertTrue(
    fbTempSensor.FFO.i_xOK,
    'Faulted with temp below threshold',
);

fbTempSensor.fFaultThreshold := 10;
fbTempSensor.bVeto := FALSE;
SetTempAndRunFB(150);
AssertFalse(
    fbTempSensor.FFO.i_xOK,
    'Did not fault with temp above threshold',
);

fbTempSensor.fFaultThreshold := 5;
fbTempSensor.bVeto := TRUE;
SetTempAndRunFB(1000);
AssertTrue(
    fbTempSensor.FFO.i_xOK,
    'Faulted with manual veto',
);

TEST_FINISHED();
END_METHOD

END_FUNCTION_BLOCK

// ---- POUs/FB_FDQ_FlowMeter.TcPOU
FUNCTION_BLOCK FB_FDQ_FlowMeter
VAR_INPUT
    // Connect this input to the terminal
    iRaw AT %I*: INT;
    // The number of bits correlated with the terminal's max value. This is not necessarily the resolution parameter.
    iTermBits: UINT := 15;
    // The fReal value correlated with the terminal's max value
    fTermMax: LREAL := 60;
    // The fReal value correlated with the terminal's min value
    fTermMin: LREAL := 0;
    // Value to scale the end result to
    fResolution : LREAL := 1;
    fOffset : LREAL;
END_VAR
VAR_OUTPUT
    {attribute 'pytmc' := '
        pv: FWM
        field: EGU lpm
    '}
    fbFlowMeter : FB_AnalogInput;
END_VAR
VAR
END_VAR

fbFlowMeter(iRaw := iRaw,
iTermBits:=iTermBits,
fTermMax:=fTermMax,
fTermMin:=fTermMin,
fResolution:=fResolution,
fOffset:=fOffset
);

END_FUNCTION_BLOCK
